FUNCTION_BLOCK NeredaMetalSaltDosing (* CAT Function Block Type *)
  (* Standard: 61499-2 *)
  (* Version 0.0, 7/9/2026, Schneider Electric, template *)
  PACKAGE SE.Nereda;
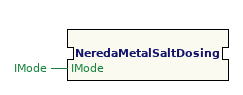
  SOCKETS
    IMode : IMode;
  END_SOCKETS
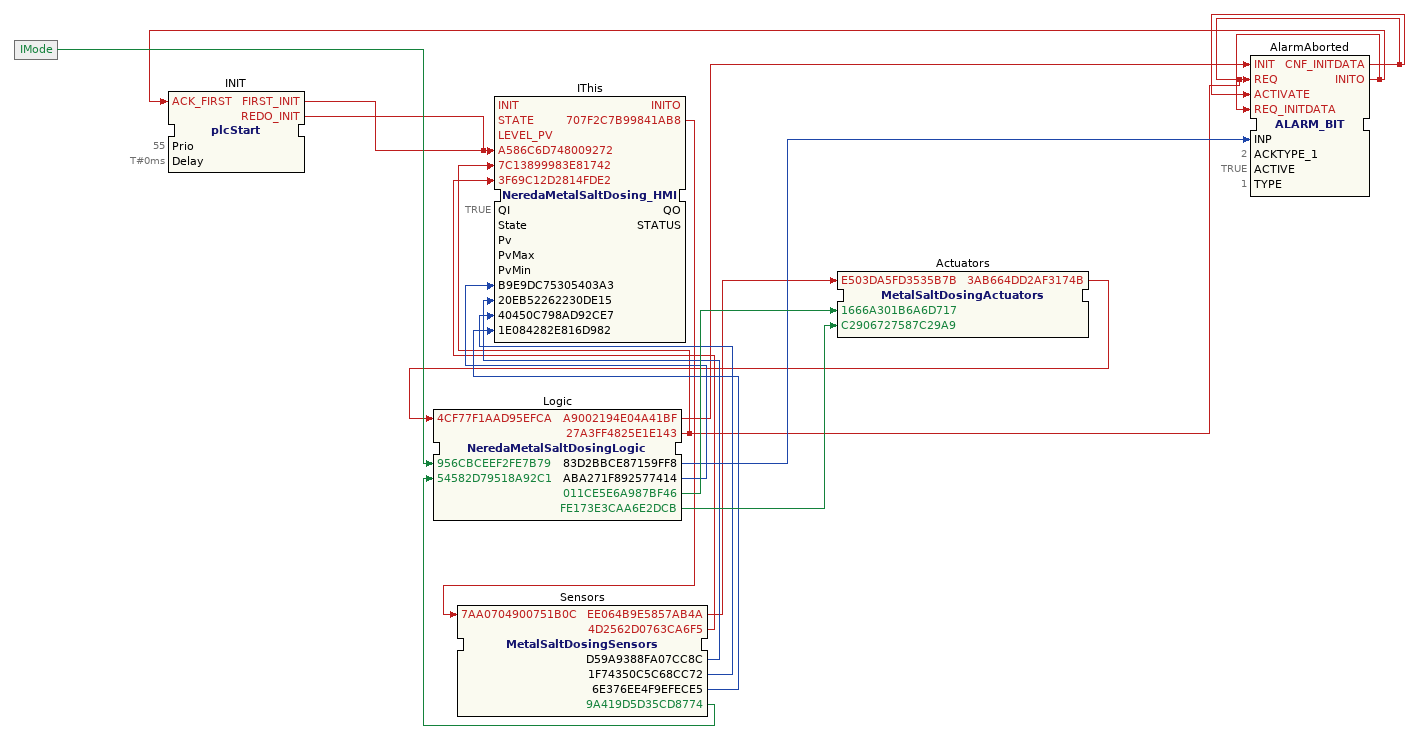
  (* 01 - FUNCTIONNAL INPUT INTERFACE *)
  (* 00 - INITIALIZATION *)
  (* 05 - LOGIC *)
  (* 06 - HMI INTERFACE *)
  (* 03 - FIELD INTERFACE *)
  (* 02 - FUNCTIONNAL OUTPUT INTERFACE *)
  (* Reactor Logic *)
  (* 04 - CHILDREN *)
  (* 4A - TYPICALS *)
  (* 07- REACTOR ALARM *)
  FBS
    INIT : plcStart(Prio := 55, Delay := T#0ms);
    IThis : NeredaMetalSaltDosing_HMI(QI := TRUE);
    Sensors : MetalSaltDosingSensors;
    Actuators : MetalSaltDosingActuators;
    Logic : NeredaMetalSaltDosingLogic;
    AlarmAborted : ALARM_BIT(ACKTYPE_1 := 2, ACTIVE := TRUE, TYPE := 1);
  END_FBS
  EVENT_CONNECTIONS
    Sensors.EE064B9E5857AB4A TO Actuators.E503DA5FD3535B7B;
    Actuators.3AB664DD2AF3174B TO Logic.4CF77F1AAD95EFCA;
    Logic.A9002194E04A41BF TO AlarmAborted.INIT;
    AlarmAborted.CNF_INITDATA TO AlarmAborted.REQ;
    AlarmAborted.CNF_INITDATA TO AlarmAborted.ACTIVATE;
    AlarmAborted.INITO TO AlarmAborted.REQ_INITDATA;
    AlarmAborted.INITO TO INIT.ACK_FIRST;
    Logic.27A3FF4825E1E143 TO AlarmAborted.REQ;
    INIT.FIRST_INIT TO IThis.A586C6D748009272;
    INIT.REDO_INIT TO IThis.A586C6D748009272;
    Logic.27A3FF4825E1E143 TO IThis.7C13899983E81742;
    Sensors.4D2562D0763CA6F5 TO IThis.3F69C12D2814FDE2;
    IThis.707F2C7B99841AB8 TO Sensors.7AA0704900751B0C;
  END_CONNECTIONS
  DATA_CONNECTIONS
    Logic.83D2BBCE87159FF8 TO AlarmAborted.INP;
    Logic.ABA271F892577414 TO IThis.B9E9DC75305403A3;
    Sensors.D59A9388FA07CC8C TO IThis.20EB52262230DE15;
    Sensors.1F74350C5C68CC72 TO IThis.40450C798AD92CE7;
    Sensors.6E376EE4F9EFECE5 TO IThis.1E084282E816D982;
  END_CONNECTIONS
  ADAPTER_CONNECTIONS
    IMode TO Logic.956CBCEEF2FE7B79;
    Sensors.9A419D5D35CD8774 TO Logic.54582D79518A92C1;
    Logic.011CE5E6A987BF46 TO Actuators.1666A301B6A6D717;
    Logic.FE173E3CAA6E2DCB TO Actuators.C2906727587C29A9;
  END_CONNECTIONS
END_FUNCTION_BLOCK
